// LS Electric XG5000 project: ABC
// PLC LSPLC

PROGRAM NewProgram (task: 스캔 프로그램)

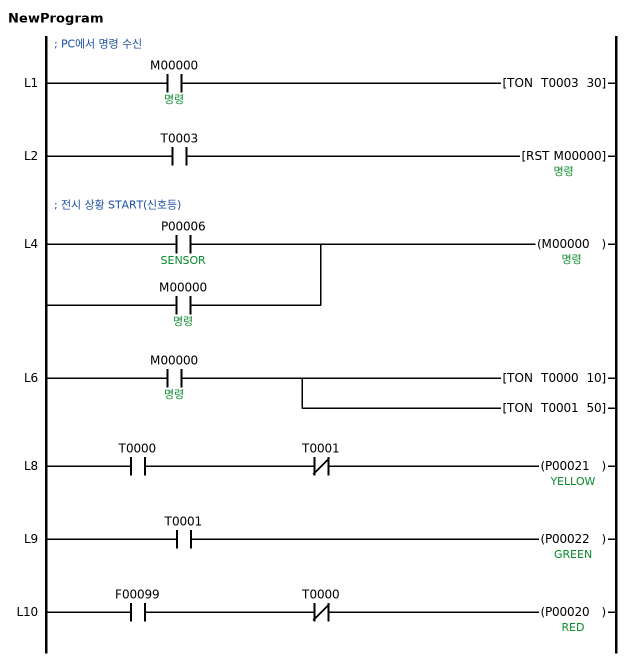
//  PC에서 명령 수신
; L1
LOAD      M00000	// 명령
TON       T0003 30
; L2
LOAD      T0003
RST       M00000	// 명령
//  전시 상황 START(신호등)
; L4
LOAD      P00006	// SENSOR
OR        M00000	// 명령
OUT       M00000	// 명령
; L6
LOAD      M00000	// 명령
TON       T0000 10
TON       T0001 50
; L8
LOAD      T0000
AND NOT   T0001
OUT       P00021	// YELLOW
; L9
LOAD      T0001
OUT       P00022	// GREEN
; L10
LOAD      F00099
AND NOT   T0000
OUT       P00020	// RED

VARIABLES AND COMMENTS (devices not used above)
D00000	WORD	CO
M00001	BIT	출력